// TIA Portal V17 export
// export: Created 2025-06-26T06:49:11.0739517Z, ExportSetting WithDefaults, DisplayName Totally Integrated Automation Portal, DisplayVersion V17 Update 8, DisplayName TIA Portal Openness, DisplayVersion V17 Update 8, DisplayName TIA Portal Version Control Interface, DisplayVersion V17, DisplayName STEP 7 Professional, DisplayVersion V17 Update 8, DisplayName STEP 7 Safety, DisplayVersion V17 Update 6, DisplayName WinCC Advanced, DisplayVersion V17 Update 8
FUNCTION_BLOCK "InverterDriveProcessing"   // FB12, FBD
TITLE = Inverter drive processing
{ S7_Optimized_Access := 'FALSE' }
AUTHOR : Heaten
VERSION : 0.1
// Command and status
// stored: AutoNumber true, IsIECCheckEnabled false, SetENOAutomatically false, UDAEnableTagReadback false
   VAR
      HBL_SC_02 { ExternalAccessible := 'False'; ExternalVisible := 'False'; ExternalWritable := 'False'} : "fbACS880";
      HBL_SC_03 { S7_SetPoint := 'True'} : "fbACS880";
      HBL_SC_01 { ExternalAccessible := 'False'; ExternalVisible := 'False'; ExternalWritable := 'False'} : "fbACS880";
      HBL_SC_10 { ExternalAccessible := 'False'; ExternalVisible := 'False'; ExternalWritable := 'False'} : "fbACS880";
   END_VAR
   VAR DB_SPECIFIC
      State : Array[0..7] of Bool;   // Profinet online state (1 bit per node)
      RetVal { ExternalAccessible := 'False'; ExternalVisible := 'False'; ExternalWritable := 'False'} : Int;   // Error code internal to DeviceStates
   END_VAR
BEGIN

REGION Network 1: Comm status all Profinet devices
   // Mode 1 = IO devices are configured
   // Mode 2 = IO devices are faulty
   // Mode 3 = IO devices are disabled
   // Mode 4 = IO devices exist
   // Mode 5 = IO devices for which a problem has occurred
   // online state bit corresponds to "Profinet device number" -> CHECK THIS IN DEVICE CONFIGURATION
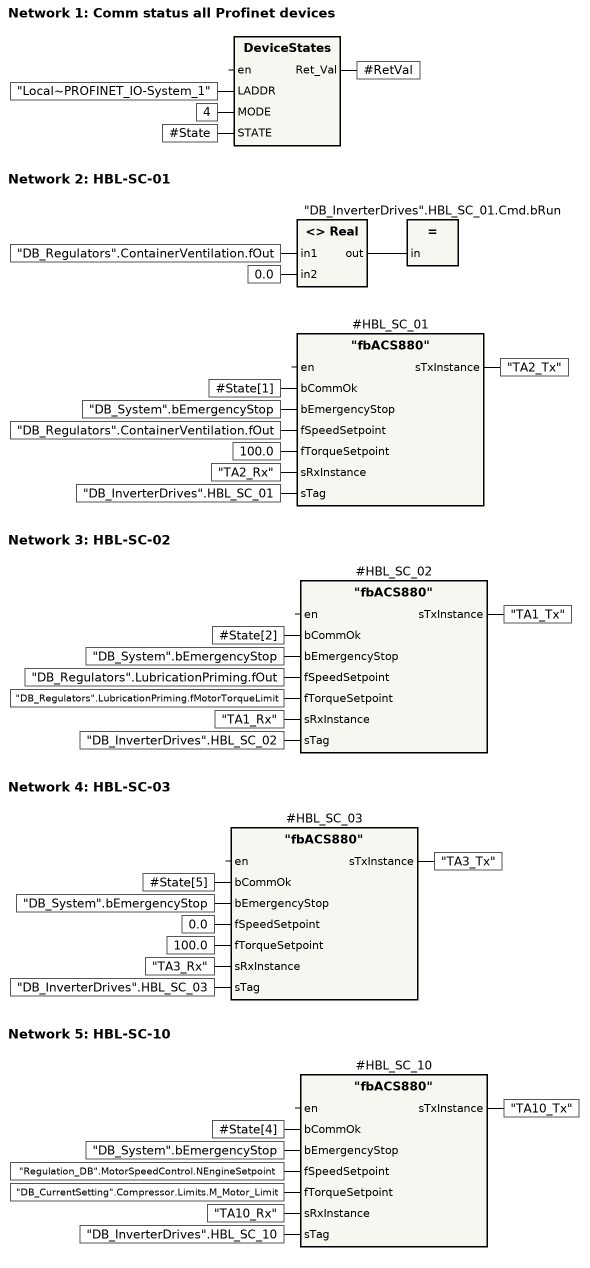
   #RetVal := DeviceStates(LADDR := "Local~PROFINET_IO-System_1", MODE := 4, STATE := #State);
END_REGION

REGION Network 2: HBL-SC-01
   "DB_InverterDrives".HBL_SC_01.Cmd.bRun := "DB_Regulators".ContainerVentilation.fOut <> 0.0;
   #HBL_SC_01(bCommOk := #State[1],   // "fbACS880"
              bEmergencyStop := "DB_System".bEmergencyStop,
              fSpeedSetpoint := "DB_Regulators".ContainerVentilation.fOut,
              fTorqueSetpoint := 100.0,
              sRxInstance := "TA2_Rx",
              sTag := "DB_InverterDrives".HBL_SC_01,
              sTxInstance => "TA2_Tx");
END_REGION

REGION Network 3: HBL-SC-02
   #HBL_SC_02(bCommOk := #State[2],   // "fbACS880"
              bEmergencyStop := "DB_System".bEmergencyStop,
              fSpeedSetpoint := "DB_Regulators".LubricationPriming.fOut,
              fTorqueSetpoint := "DB_Regulators".LubricationPriming.fMotorTorqueLimit,
              sRxInstance := "TA1_Rx",
              sTag := "DB_InverterDrives".HBL_SC_02,
              sTxInstance => "TA1_Tx");
END_REGION

REGION Network 4: HBL-SC-03
   #HBL_SC_03(bCommOk := #State[5],   // "fbACS880"
              bEmergencyStop := "DB_System".bEmergencyStop,
              fSpeedSetpoint := 0.0,
              fTorqueSetpoint := 100.0,
              sRxInstance := "TA3_Rx",
              sTag := "DB_InverterDrives".HBL_SC_03,
              sTxInstance => "TA3_Tx");
END_REGION

REGION Network 5: HBL-SC-10
   #HBL_SC_10(bCommOk := #State[4],   // "fbACS880"
              bEmergencyStop := "DB_System".bEmergencyStop,
              fSpeedSetpoint := "Regulation_DB".MotorSpeedControl.NEngineSetpoint,
              fTorqueSetpoint := "DB_CurrentSetting".Compressor.Limits.M_Motor_Limit,
              sRxInstance := "TA10_Rx",
              sTag := "DB_InverterDrives".HBL_SC_10,
              sTxInstance => "TA10_Tx");
END_REGION
END_FUNCTION_BLOCK
